// TIA Portal V17 export
// export: Created 2026-04-13T11:12:42.2607674Z, ExportSetting WithDefaults, DisplayName Totally Integrated Automation Portal, DisplayVersion V17 Update 4, DisplayName TIA Portal Openness, DisplayVersion V17 Update 4, DisplayName TIA Portal Version Control Interface, DisplayVersion V17, DisplayName SINAMICS Startdrive Advanced, DisplayVersion V17, DisplayName SINAMICS Startdrive G130, G150, S120, S150, SINAMICS MV, S210, DisplayVersion V17, DisplayName SINAMICS Startdrive G110M, G120, G120C, G120D, G120P, G115D, DisplayVersion V17, DisplayName STEP 7 Professional, DisplayVersion V17 Update 4, DisplayName STEP 7 Safety, DisplayVersion V17, DisplayName WinCC Professional, DisplayVersion V17 Update 4
FUNCTION_BLOCK "0-模拟量输入"   // FB35, SCL
{ S7_Optimized_Access := 'TRUE' }
VERSION : 0.1
// stored: AutoNumber true, IsIECCheckEnabled false, IsRetainMemResEnabled false, MemoryReserve 100, SetENOAutomatically false, UDAEnableTagReadback false
   VAR_INPUT
      模拟量数据输入 : Int;
      上限模拟 : Real := 27648.0;
      下限模拟 : Real := 5530.0;
      上限工程 : Real := 100.0;
      下限工程 : Real := 0.0;
      修正值 : Real;
      错误确认 : Bool;
      高高限工程量 : Real := 90.0;
      高限工程量 : Real := 80.0;
      低限工程量 : Real := 20.0;
      低低限工程量 : Real := 10.0;
      高高限位滤波时间设定 : Time := T#1s;
      高限位滤波时间设定 : Time := T#1s;
      低限位滤波时间设定 : Time := T#1s;
      低低限位滤波时间设定 : Time := T#1s;
      MODE : Byte := 16#1;   // 0报警输出不自动消除，1报警情况结束自动消除 2.高高或低低限位保持报警，其余自动确认报警
   END_VAR
   VAR_OUTPUT
      工程量数据输出 : Real;
      断线错误 : Bool;
      超过高高限位 : Bool;
      超过高限位 : Bool;
      低于低限位 : Bool;
      低于低低限位 : Bool;
   END_VAR
   VAR
      临时模拟量数据输入 : Real;
      缩放比例 : Real;
      T : Struct
         高高限位滤波时间 { S7_SetPoint := 'True'} : TON_TIME;
         高限位滤波时间 { S7_SetPoint := 'True'} : TON_TIME;
         低限位滤波时间 { S7_SetPoint := 'True'} : TON_TIME;
         低低限位滤波时间 { S7_SetPoint := 'True'} : TON_TIME;
      END_STRUCT;
   END_VAR
BEGIN
   #临时模拟量数据输入 := INT_TO_REAL(#模拟量数据输入);  //将模拟量输入转换为real类型
   // IF #临时模拟量数据输入 > #模拟量Max THEN
   //     #临时模拟量数据输入 := #模拟量Max;
   // END_IF;
   // IF #临时模拟量数据输入 < #模拟量Min THEN
   //     #临时模拟量数据输入 := #模拟量Min;
   // END_IF;
   #缩放比例 := (#上限工程 - #下限工程) / (#上限模拟 - #下限模拟);//算出实际值与模拟量的缩放比例
   #工程量数据输出 := (#模拟量数据输入 - #下限模拟) * #缩放比例 + #下限工程+#修正值;      //转换完成


   //2
   //
   IF (#临时模拟量数据输入 > 30000 OR #临时模拟量数据输入 < 4000 )
       AND NOT #错误确认 THEN
       #断线错误 := 1;
   ELSE
       #断线错误 := 0;
   END_IF;

   //3
   //

   #T.高高限位滤波时间(IN := #工程量数据输出 > #高高限工程量,
               PT := #高高限位滤波时间设定);
   IF #T.高高限位滤波时间.Q OR (#超过高高限位 AND (#MODE = 0 OR #MODE = 2)) AND NOT #错误确认 THEN

       #超过高高限位 := 1;
   ELSE
       #超过高高限位 := 0;
   END_IF;

   (* IF #超过高高限位 AND (#MODE = 0 OR #MODE = 2) AND NOT #错误确认 THEN
       #超过高高限位 := 1;
   ELSE
       #超过高高限位 := 0;
   END_IF; *)

   //4
   //
   #T.高限位滤波时间(IN := #工程量数据输出 >= #高限工程量,
              PT := #高限位滤波时间设定);
   IF #T.高限位滤波时间.Q OR (#超过高限位 AND #MODE = 0) AND NOT #错误确认 THEN
       #超过高限位 := 1;
   ELSE
       #超过高限位 := 0;
   END_IF;

   //5
   //
   #T.低限位滤波时间(IN := #工程量数据输出 <= #低限工程量,
              PT := #低限位滤波时间设定);

   IF #T.低限位滤波时间.Q OR (#低于低限位 AND #MODE = 0) AND NOT #错误确认 THEN
       #低于低限位 := 1;
   ELSE
       #低于低限位 := 0;
   END_IF;

   (* IF #低于低限位 AND #MODE=0 THEN
       #低于低限位 := 1;
   ELSE
       #低于低限位 := 0;
   END_IF; *)

   //6
   //
   #T.低低限位滤波时间(IN := #工程量数据输出 <= #低低限工程量,
               PT := #低低限位滤波时间设定);
   IF #T.低低限位滤波时间.Q OR (#低于低低限位 AND (#MODE = 0 OR #MODE = 2)) AND NOT #错误确认 THEN
       #低于低低限位 := 1;
   ELSE
       #低于低低限位 := 0;
   END_IF;

   (* IF #低于低低限位 AND (#MODE=0 OR #MODE=2) AND NOT #错误确认  THEN
       #低于低低限位 := 1;
   ELSE
       #低于低低限位 := 0;
   END_IF; *)
END_FUNCTION_BLOCK
